// TIA Portal project "Proyecto3" (V16)

(* hardware
DEVICE "S7-1200 station_1"  S7-1200 Station
   slot 0: "Rack_0"  S7-1200 Rack  Rack  V1.0
   slot 1: "PLC_1"  CPU 1214C AC/DC/Rly  6ES7 214-1BG40-0XB0  V4.4
*)

// ===== PLC "PLC_1"  CPU 1214C AC/DC/Rly =====

VAR_GLOBAL   // PLC tag table "Tabla de variables estándar"
   "Tag_1" AT %I0.0 : Bool;
   "Tag_2" AT %I0.1 : Bool;
   "Tag_3" AT %Q0.0 : Bool;
END_VAR

FUNCTION_BLOCK "Bloque_1"   // FB1, LAD
{ S7_Optimized_Access := 'TRUE' }
VERSION : 0.1
BEGIN
END_FUNCTION_BLOCK

FUNCTION "Bloque_2" : Void   // FC1, LAD
{ S7_Optimized_Access := 'TRUE' }
VERSION : 0.1
BEGIN

REGION Network 1
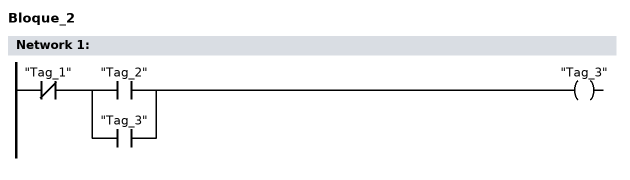
   RUNG wire#powerrail
      I_Contact( "Tag_1" )
      wire#w1
      Contact( "Tag_2" )
      wire#w2
      Coil( "Tag_3" )
   END_RUNG
   RUNG wire#w1
      Contact( "Tag_3" )
   END_RUNG wire#w2
   // the same network as SCL:
   "Tag_3" := NOT "Tag_1" AND ("Tag_2" OR "Tag_3");
END_REGION
END_FUNCTION

ORGANIZATION_BLOCK "Main"   // OB1, LAD, ProgramCycle
TITLE = "Main Program Sweep (Cycle)"
{ S7_Optimized_Access := 'TRUE' }
VERSION : 0.1
   VAR_INPUT
      Initial_Call : Bool;   // Initial call of this OB
      Remanence : Bool;   // =True, if remanent data are available
   END_VAR
BEGIN

REGION Network 1
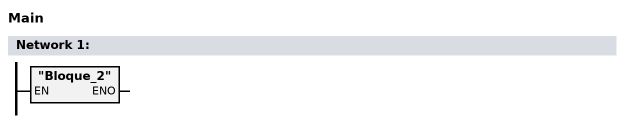
   RUNG wire#powerrail
      "Bloque_2"()
   END_RUNG
   // the same network as SCL:
   "Bloque_2"();
END_REGION
END_ORGANIZATION_BLOCK